Universal Robots PolyScope program: h13.urp

Program h13 (installation=default directory=/programs createdIn=5.4.3.76201 lastSavedIn=5.4.3.76201 robotSerialNumber=20195001485)
Calibrated DH parameters: a=[0.000123, -0.611833, -0.350641, 0.000064, -0.000085, 0]; d=[0.18107, -11.986108, 254.021851, -241.861392, 0.119787, 0.115693]; alpha=[1.570574, 0.001664, -0.001863, 1.570661, -1.570447, 0]; deltaTheta=[0, -0.032583, -0.877293, 0.909879, 0.000002, 0]
Robot Program (runOnlyOnce=true)
  MoveJ speed 60 deg/s, acceleration 80 deg/s^2 (useActiveTCP=true) feature=Base
    Waypoint Waypoint_1: TCP in base x=433.025 y=-467.959 z=522.311 mm, rx=1.5003 ry=0.5214 rz=0.531 rad; joints [114.262, -95.596, 110.756, -15.575, 75.682, 0.208] deg
    URCap Gripper (Robotiq_Grippers, Robotiq Inc.) dataModel(position=0.0, force=0.0, speed=0.0, positionInDouble=0.0, forceInDouble=0.0, speedInDouble=0.0, slaveIds=[9], blocking=true)
    Waypoint Waypoint_2: TCP in base x=537.105 y=-592.669 z=524.349 mm, rx=1.5003 ry=0.5215 rz=0.531 rad; joints [118.086, -79.882, 94.136, -14.675, 79.502, 0.206] deg
    URCap Gripper (Robotiq_Grippers, Robotiq Inc.) dataModel(position=100.0, force=0.0, speed=0.0, positionInDouble=100.0, forceInDouble=0.0, speedInDouble=0.0, slaveIds=[9], blocking=true)
    Waypoint Waypoint_1: TCP in base x=433.025 y=-467.959 z=522.311 mm, rx=1.5003 ry=0.5214 rz=0.531 rad; joints [114.262, -95.596, 110.756, -15.575, 75.682, 0.208] deg
